VAR_GLOBAL
	Elevator:FB_Elevator;
	Floors:ARRAY[1..4]	OF	ST_Floor;
	RequestedFloor: INT;
	ActualFloor: INT;
END_VAR

(* stored: Version 1.1.0.1, ProductVersion 3.1.4024.11
   GVL GVL: Id {b29cab17-c559-4e76-9865-572eff242459} *)
